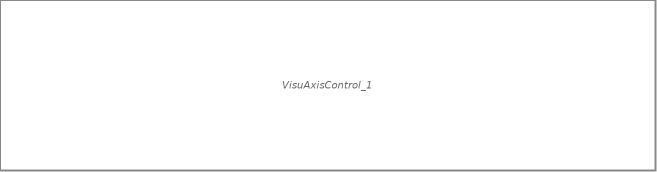
VISUALIZATION VisuAxisY_1  // 657x172
    Frame (0,0 655x170)
        shows VisuAxisControl_1(sAxisName_1 := sAxisYName, stAxisVisu_1 := stAxisY)
END_VISUALIZATION

(* stored: Version 1.1.0.1, ProductVersion 3.1.4022.6
   Visu VisuAxisY_1: Id {0390e8cd-e7f4-4e08-a713-fc02944b2c22} *)
